Universal Robots URScript: T011_qwen2.5-coder_32b_baseline_rep1_retry3.urscript

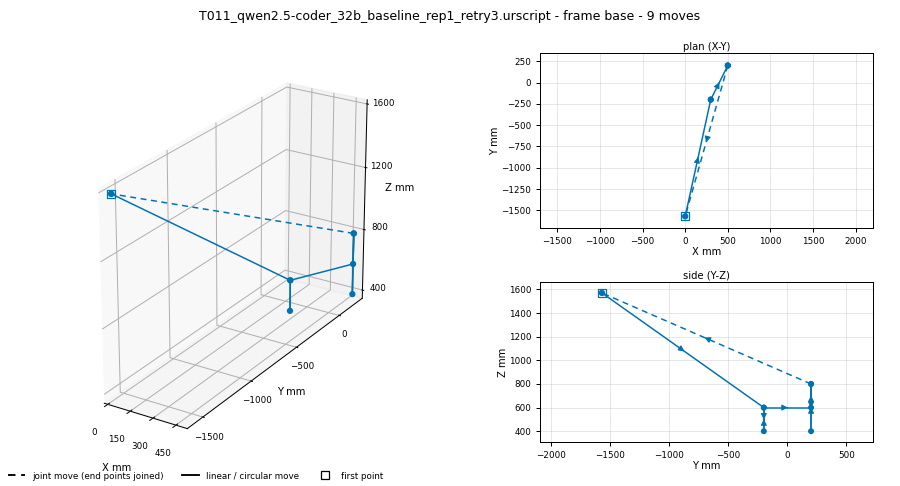
[picture p0: tool path of T011_qwen2.5-coder_32b_baseline_rep1_retry3.urscript in frame base, 9 of 9 moves have a stored position in this frame; points joined in program order, loops and branches not executed]
def dual_zone_pick_place():
    # Set payload
    set_payload(1.2)

    # Home position
    movej(p[0.0, -1.5708, 1.5708, -1.5708, -1.5708, 0.0], a=1.4, v=1.05)

    # Above storage bin
    movel(p[0.3, -0.2, 0.6, 2.2, 2.2, 0.0], a=1.2, v=0.28)

    # Descend to pick
    movel(p[0.3, -0.2, 0.4, 2.2, 2.2, 0.0], a=1.2, v=0.12)

    # Lift from bin
    movel(p[0.3, -0.2, 0.6, 2.2, 2.2, 0.0], a=1.2, v=0.2)

    # Transit to handoff zone
    movel(p[0.5, 0.2, 0.6, 2.2, 2.2, 0.0], a=1.2, v=0.25)

    # Above handoff zone (additional move)
    movel(p[0.5, 0.2, 0.8, 2.2, 2.2, 0.0], a=1.2, v=0.3)

    # Descend to place
    movel(p[0.5, 0.2, 0.4, 2.2, 2.2, 0.0], a=1.2, v=0.12)

    # Lift from handoff zone (additional move)
    movel(p[0.5, 0.2, 0.8, 2.2, 2.2, 0.0], a=1.2, v=0.3)

    # Return to home
    movej(p[0.0, -1.5708, 1.5708, -1.5708, -1.5708, 0.0], a=1.4, v=1.05)

end

# Execute the function
dual_zone_pick_place()
